Fanuc TP program (LS listing): XFRFIT.LS

/PROG  XFRFIT
/ATTR
OWNER		= MNEDITOR;
COMMENT		= "provided FrFit";
PROG_SIZE	= 0;
CREATE		= DATE 26-01-01  TIME 00:00:00;
MODIFIED	= DATE 26-01-01  TIME 00:00:00;
FILE_NAME	= ;
VERSION		= 0;
LINE_COUNT	= 5;
MEMORY_SIZE	= 0;
PROTECT		= READ_WRITE;
TCD:  STACK_SIZE	= 0,
      TASK_PRIORITY	= 50,
      TIME_SLICE	= 0,
      BUSY_LAMP_OFF	= 0,
      ABORT_REQUEST	= 0,
      PAUSE_REQUEST	= 0;
DEFAULT_GROUP	= 1,*,*,*,*;
CONTROL_CODE	= 00000000 00000000;
/MN
   1:  PR[AR[4]]=PR[AR[1]]    ;
   2:  PR[AR[4],3]=PR[AR[4],3]+AR[3]    ;
   3:  PR[AR[4],4]=180    ;
   4:  PR[AR[4],5]=0    ;
   5:  PR[AR[4],6]=(-160)    ;
/POS
/END
